# EPICS IOC start-up script: examples/test/PSI/EP7211-0034_AM8111/EP7211-0034_AM8111_CSP.iocsh
require ecmccfg v7_RC1

${SCRIPTEXEC} ${ecmccfg_DIR}configureSlave.cmd, "SLAVE_ID=3, HW_DESC=EP7211-0034_CSP, CONFIG=-Motor-Beckhoff-AM8111-0F20-0000"

epicsEnvSet("DEV",      "STEST-MYDEVICE")
${SCRIPTEXEC} ${ecmccfg_DIR}configureAxis.cmd,            "CONFIG=./cfg/AM8111_CSP.pax"
